INTERFACE I_Handler

METHOD PUBLIC M_Request
VAR_INPUT
	stEvent:			ST_Event;
END_VAR
END_METHOD

PROPERTY PUBLIC P_Next : I_Handler
GET
END_GET
SET
END_SET
END_PROPERTY

END_INTERFACE

(* stored: Version 1.1.0.1, ProductVersion 3.1.4024.12
   Itf I_Handler: Id {76c924fb-9512-49da-9ecf-f9832661e458}
   Method M_Request: Id {a20fe26c-2355-4f10-b0a3-ae027dfea6fe}
   Property P_Next: Id {48611710-ff4c-4320-a1e6-09e5151902e2}
   Get Get: Id {23236f31-1abe-42e1-b70f-a139733fd44f}
   Set Set: Id {45804c4f-a0a1-4b87-b396-4a6ed6ee4597} *)
